Yaskawa INFORM job: SYS_RESET_CELL.JBI

/JOB
//NAME SYS_RESET_CELL
//POS
///NPOS 0,0,0,0,0,0
//INST
///DATE 2021/12/03 00:22
///ATTR SC,RW
///GROUP1 RB1
NOP
CALL JOB:SYS_SPINDE_OFF
CALL JOB:SYS_STOP_FILTERS
DOUT OT#(19) OFF
END
